{attribute 'qualified_only'}
{attribute 'strict'}
TYPE StackerBeltTableMode :
(
	Mode_Standard	:= 0,
	Mode_Manual		:= 1,
	Mode_Simulation	:= 2
	
);
END_TYPE

(* stored: Version 1.1.0.1, ProductVersion 3.1.4024.12
   DUT StackerBeltTableMode: Id {619875af-b90c-4cdc-8ed1-12c6eeaf8b3b} *)
